// TwinCAT 3 PLC project SLAC_19046_PLC_v2
// ProgramVersion: 3.1.4023.0
// libraries:
//   Tc2_MC2, * (Beckhoff Automation GmbH)
//   Tc2_Standard, * (Beckhoff Automation GmbH)
//   Tc2_System, * (Beckhoff Automation GmbH)
//   Tc2_Utilities, * (Beckhoff Automation GmbH)
//   Tc3_Module, * (Beckhoff Automation GmbH)
// project tree:
//   / PlcTask.TcTTO
//   POUs/ AirPitch_Limit_Switches.TcPOU, AirRoll_Limit_Switches.TcPOU, AirVertical_Limit_Switches.TcPOU, CrystalGap_Limit_Switches.TcPOU, FB_Test.TcPOU, MAIN.TcPOU, YAG_LimitSwitched.TcPOU
// real-time tasks:
//   TASK PlcTask: cycle T#10ms, priority 20, ADS port 350
// motion (NC):
//   TASK NC-Task 1 SAF: cycle T#2ms, priority 4, ADS port 501
//   TASK NC-Task 1 SVB: cycle T#10ms, priority 8, ADS port 511
//   AXIS AirPitch (id 1)
//     General: UnitName=mrad
//     Dynamic: Acceleration=8.99313, Deceleration=8.99313, Jerk=27.7544
//     Velo: SlowManual=1, FastManual=2, Maximum=3.1
//     TargetPosControl: Range=0.001
//     OtherSettings: AllowMotionCmdToSlave=true, PulseDistancePos=0.5, PulseDistanceNeg=0.5
//     encoder EncType=29
//       EncPara: ScaleFactorNumerator=1.2657e-07, Offset=-4.6852, MaxCount=#xffffffff, ReferenceSystem=1
//         SoftEndMinControl: Enable=true, Range=-3.5
//         SoftEndMaxControl: Enable=true, Range=2.8
//         Inc: RefSoftSyncMask=#x0000ffff
//     drive DrvType=24
//       DrvPara: Inverse=true
//         Analog: VeloReferenz=3.3, TorqueSetpointScale=10, ScaleFactorActTorque=0.1
//         TimeComp: TaskDelayCycles=1
//     controller CtrType=3
//       CtrPara: PriorControlFactor=1
//         PosDiffControl: Range=0.5
//         PID: PosKp=10, PosTv=0.2, DeadBandPosition=0.0001
//         Observer: BandWidth=20
//   AXIS AirVert (id 2)
//     Dynamic: Acceleration=2.95205, Deceleration=2.95205, Jerk=8.98412
//     Velo: SlowManual=0.1, FastManual=0.3, Maximum=1
//     PositionAreaControl: Range=0.05
//     TargetPosControl: Range=0.0001
//     OtherSettings: AllowMotionCmdToSlave=true
//     encoder EncType=29
//       EncPara: ScaleFactorNumerator=1e-06, Offset=-10.712, MaxCount=#xffffffff
//         SoftEndMinControl: Enable=true, Range=-4.1
//         SoftEndMaxControl: Enable=true, Range=3
//         Inc: RefSoftSyncMask=#x0000ffff
//     drive DrvType=24
//       DrvPara: Inverse=true
//         Analog: VeloReferenz=3, TorqueSetpointScale=10, ScaleFactorActTorque=0.1
//         TimeComp: TaskDelayCycles=1
//     controller CtrType=3
//       CtrPara: PriorControlFactor=1
//         PosDiffControl: Range=0.15
//         PID: PosKp=7, PosTv=0.2
//         Observer: BandWidth=20
//   AXIS AirRoll (id 3)
//     General: UnitName=mrad
//     Dynamic: Acceleration=0.424188, Deceleration=0.424188, Jerk=6.42628
//     Velo: SlowManual=0.3, FastManual=1, Maximum=2.8
//     PositionAreaControl: Range=0.2
//     TargetPosControl: Range=0.0005
//     OtherSettings: AllowMotionCmdToSlave=true, PulseDistancePos=1, PulseDistanceNeg=1
//     encoder EncType=29
//       EncPara: ScaleFactorNumerator=2.4267e-07, Offset=-1031.2195, MaxCount=#xffffffff
//         SoftEndMinControl: Enable=true, Range=-4.8
//         SoftEndMaxControl: Enable=true, Range=6.1
//         Inc: RefSoftSyncMask=#x0000ffff
//     drive DrvType=24
//       Analog: VeloReferenz=3, TorqueSetpointScale=10, ScaleFactorActTorque=0.1
//       TimeComp: TaskDelayCycles=1
//     controller CtrType=3
//       CtrPara: PriorControlFactor=1
//         PosDiffControl: Range=0.5
//         PID: PosKp=10, PosTv=0.2, DeadBandPosition=0.0001
//         Observer: BandWidth=20
//   AXIS CrystalGap (id 4)
//     Dynamic: Acceleration=1.59597, Deceleration=1.59597, Jerk=4.61435
//     Velo: SlowManual=0.075, FastManual=0.2, Maximum=0.6
//     PositionAreaControl: Range=0.01
//     TargetPosControl: Range=0.0001
//     OtherSettings: AllowMotionCmdToSlave=true, PulseDistancePos=0.05, PulseDistanceNeg=0.05
//     encoder EncType=29
//       EncPara: ScaleFactorNumerator=1e-06, Offset=-19.5127, MaxCount=#xffffffff
//         SoftEndMinControl: Enable=true, Range=0.05
//         SoftEndMaxControl: Enable=true, Range=9.1
//         Inc: RefSoftSyncMask=#x0000ffff
//     drive DrvType=24
//       DrvPara: Inverse=true
//         Analog: VeloReferenz=0.3, TorqueSetpointScale=10, ScaleFactorActTorque=0.1
//         TimeComp: TaskDelayCycles=1
//     controller CtrType=3
//       CtrPara: PriorControlFactor=1
//         PosDiffControl: Range=0.15
//         PID: PosKp=4, PosTv=0.2, PosTd=1, DeadBandPosition=0.0001
//         Observer: BandWidth=20
//   AXIS YAG (id 5)
//     Dynamic: Acceleration=4.26689, Deceleration=4.26689, Jerk=19.1646
//     Velo: SlowManual=0.5, FastManual=1, Maximum=2
//     PositionAreaControl: Range=0.05
//     TargetPosControl: Range=0.05
//     OtherSettings: AllowMotionCmdToSlave=true
//     encoder EncType=29
//       EncPara: ScaleFactorNumerator=1e-06, Offset=-17, MaxCount=#xffffffff
//         SoftEndMinControl: Enable=true, Range=-0.53
//         SoftEndMaxControl: Enable=true, Range=41.6
//         Inc: RefSoftSyncMask=#x0000ffff
//     drive DrvType=24
//       Analog: VeloReferenz=20, TorqueSetpointScale=10, ScaleFactorActTorque=0.1
//       TimeComp: TaskDelayCycles=1
//     controller CtrType=3
//       CtrPara: PriorControlFactor=1
//         PosDiffControl: Range=1
//         PID: PosKp=15, PosTv=0.2, DeadBandPosition=0.01
//         Observer: BandWidth=20
//   AXIS Test (id 6)
//     TargetPosControl: Range=0.01
//     OtherSettings: AllowMotionCmdToSlave=true
//     encoder EncType=1
//     drive DrvType=5
//       Analog: TorqueSetpointScale=10, ScaleFactorActTorque=0.1
//       TimeComp: TaskDelayCycles=1
//     controller CtrType=1
//       CtrPara: PriorControlFactor=1
//         Observer: BandWidth=20
// I/O:
//   DEVICE Device 1 (EtherCAT), AmsNetId 134.79.81.23.2.1
//     Term 3 (EK1100) [EK1100 EtherCAT Coupler (2A E-Bus)]
//       Term 4 (EL7047) Air Pitch [EL7047 1Ch. Stepper motor output stage (50V, 5A)]
//       Term 5 (EL7047) Air Vertical [EL7047 1Ch. Stepper motor output stage (50V, 5A)]
//       Term 6 (EL7047) Air Roll [EL7047 1Ch. Stepper motor output stage (50V, 5A)]
//       Term 7 (EL7047) Crystal Gap [EL7047 1Ch. Stepper motor output stage (50V, 5A)]
//       Term 8 (EL7047) YAG [EL7047 1Ch. Stepper motor output stage (50V, 5A)]
//       Term 19 (EL9400) E-Bus Power Supplier [EL9400 E-Bus Power Supplier]
//       Term 9 (EL5042) Ch1 AirP Ch2 AirV [EL5042 2Ch. BiSS-C Encoder]
//       Term 10 (EL5042) Ch1 AirR Ch2 CGap [EL5042 2Ch. BiSS-C Encoder]
//       Term 11 (EL5042) Ch1 YAG [EL5042 2Ch. BiSS-C Encoder]
//       Term 13 (EL3201) Pt100 Upper Cryst [EL3201 1Ch. Ana. Input PT100 (RTD)]
//       Term 14 (EL3201) Pt100 Lower Cryst [EL3201 1Ch. Ana. Input PT100 (RTD)]
//       Term 15 (EL3201) Pt100 YAG [EL3201 1Ch. Ana. Input PT100 (RTD)]
//       Term 16 (EL3201) Pt100 Heatsink [EL3201 1Ch. Ana. Input PT100 (RTD)]
//       Term 17 (EL2634) Camera and Fan Relay [EL2634 4Ch. Relay Output, NO (250V AC / 30V DC)]
//       Term 18 (EL9011) [EL9011 End Terminal]
// variable links:
//   NC-Task 1 SAF/Axes/AirPitch <-> Device 1 (EtherCAT)/Term 3 (EK1100)/Term 4 (EL7047) Air Pitch
//     Drive/Inputs/In/nState1 @bit 3 <-> STM Status/Status/Error
//     Drive/Inputs/In/nState1 @bit 7 <-> STM Status/Status/Motor stall
//     Drive/Inputs/In/nState1 @bit 5 <-> STM Status/Status/Moving negative
//     Drive/Inputs/In/nState1 @bit 4 <-> STM Status/Status/Moving positive
//     Drive/Inputs/In/nState1 @bit 1 <-> STM Status/Status/Ready
//     Drive/Inputs/In/nState1 <-> STM Status/Status/Ready to enable
//     Drive/Inputs/In/nState1 @bit 6 <-> STM Status/Status/Torque reduced
//     Drive/Inputs/In/nState1 @bit 2 <-> STM Status/Status/Warning
//     Drive/Inputs/In/nState2 @bit 3 <-> STM Status/Status/Digital input 1
//     Drive/Inputs/In/nState2 @bit 4 <-> STM Status/Status/Digital input 2
//     Drive/Inputs/In/nState2 @bit 5 <-> STM Status/Status/Sync error
//     Drive/Inputs/In/nState2 @bit 7 <-> STM Status/Status/TxPDO Toggle
//     Drive/Inputs/In/nState4 @bit 1 <-> WcState/InputToggle
//     Drive/Inputs/In/nState4 <-> WcState/WcState
//     Drive/Outputs/Out/nCtrl1 <-> STM Control/Control/Enable
//     Drive/Outputs/Out/nCtrl1 @bit 2 <-> STM Control/Control/Reduce torque
//     Drive/Outputs/Out/nCtrl1 @bit 1 <-> STM Control/Control/Reset
//     Drive/Outputs/Out/nCtrl2 @bit 3 <-> STM Control/Control/Digital output 1
//     Drive/Outputs/Out/nDataOut2[0] <-> STM Velocity/Velocity
//   NC-Task 1 SAF/Axes/AirPitch <-> Device 1 (EtherCAT)/Term 3 (EK1100)/Term 9 (EL5042) Ch1 AirP Ch2 AirV
//     Enc/Inputs/In/nComState @bit 1 <-> WcState/InputToggle
//     Enc/Inputs/In/nComState <-> WcState/WcState
//     Enc/Inputs/In/nDataIn1 <-> FB Inputs Channel 1/Position
//     Enc/Inputs/In/nState1 @bit 12 <-> FB Inputs Channel 1/Status/Diag
//     Enc/Inputs/In/nState1 @bit 1 <-> FB Inputs Channel 1/Status/Error
//     Enc/Inputs/In/nState1 @bit 14 <-> FB Inputs Channel 1/Status/Input cycle counter
//     Enc/Inputs/In/nState1 @bit 2 <-> FB Inputs Channel 1/Status/Ready
//     Enc/Inputs/In/nState1 @bit 13 <-> FB Inputs Channel 1/Status/TxPDO State
//     Enc/Inputs/In/nState1 <-> FB Inputs Channel 1/Status/Warning
//   NC-Task 1 SAF/Axes/AirRoll <-> Device 1 (EtherCAT)/Term 3 (EK1100)/Term 10 (EL5042) Ch1 AirR Ch2 CGap
//     Enc/Inputs/In/nComState @bit 1 <-> WcState/InputToggle
//     Enc/Inputs/In/nComState <-> WcState/WcState
//     Enc/Inputs/In/nDataIn1 <-> FB Inputs Channel 1/Position
//     Enc/Inputs/In/nState1 @bit 12 <-> FB Inputs Channel 1/Status/Diag
//     Enc/Inputs/In/nState1 @bit 1 <-> FB Inputs Channel 1/Status/Error
//     Enc/Inputs/In/nState1 @bit 14 <-> FB Inputs Channel 1/Status/Input cycle counter
//     Enc/Inputs/In/nState1 @bit 2 <-> FB Inputs Channel 1/Status/Ready
//     Enc/Inputs/In/nState1 @bit 13 <-> FB Inputs Channel 1/Status/TxPDO State
//     Enc/Inputs/In/nState1 <-> FB Inputs Channel 1/Status/Warning
//   NC-Task 1 SAF/Axes/AirRoll <-> Device 1 (EtherCAT)/Term 3 (EK1100)/Term 6 (EL7047) Air Roll
//     Drive/Inputs/In/nState1 @bit 3 <-> STM Status/Status/Error
//     Drive/Inputs/In/nState1 @bit 7 <-> STM Status/Status/Motor stall
//     Drive/Inputs/In/nState1 @bit 5 <-> STM Status/Status/Moving negative
//     Drive/Inputs/In/nState1 @bit 4 <-> STM Status/Status/Moving positive
//     Drive/Inputs/In/nState1 @bit 1 <-> STM Status/Status/Ready
//     Drive/Inputs/In/nState1 <-> STM Status/Status/Ready to enable
//     Drive/Inputs/In/nState1 @bit 6 <-> STM Status/Status/Torque reduced
//     Drive/Inputs/In/nState1 @bit 2 <-> STM Status/Status/Warning
//     Drive/Inputs/In/nState2 @bit 3 <-> STM Status/Status/Digital input 1
//     Drive/Inputs/In/nState2 @bit 4 <-> STM Status/Status/Digital input 2
//     Drive/Inputs/In/nState2 @bit 5 <-> STM Status/Status/Sync error
//     Drive/Inputs/In/nState2 @bit 7 <-> STM Status/Status/TxPDO Toggle
//     Drive/Inputs/In/nState4 @bit 1 <-> WcState/InputToggle
//     Drive/Inputs/In/nState4 <-> WcState/WcState
//     Drive/Outputs/Out/nCtrl1 <-> STM Control/Control/Enable
//     Drive/Outputs/Out/nCtrl1 @bit 2 <-> STM Control/Control/Reduce torque
//     Drive/Outputs/Out/nCtrl1 @bit 1 <-> STM Control/Control/Reset
//     Drive/Outputs/Out/nCtrl2 @bit 3 <-> STM Control/Control/Digital output 1
//     Drive/Outputs/Out/nDataOut2[0] <-> STM Velocity/Velocity
//   NC-Task 1 SAF/Axes/AirVert <-> Device 1 (EtherCAT)/Term 3 (EK1100)/Term 5 (EL7047) Air Vertical
//     Drive/Inputs/In/nState1 @bit 3 <-> STM Status/Status/Error
//     Drive/Inputs/In/nState1 @bit 7 <-> STM Status/Status/Motor stall
//     Drive/Inputs/In/nState1 @bit 5 <-> STM Status/Status/Moving negative
//     Drive/Inputs/In/nState1 @bit 4 <-> STM Status/Status/Moving positive
//     Drive/Inputs/In/nState1 @bit 1 <-> STM Status/Status/Ready
//     Drive/Inputs/In/nState1 <-> STM Status/Status/Ready to enable
//     Drive/Inputs/In/nState1 @bit 6 <-> STM Status/Status/Torque reduced
//     Drive/Inputs/In/nState1 @bit 2 <-> STM Status/Status/Warning
//     Drive/Inputs/In/nState2 @bit 3 <-> STM Status/Status/Digital input 1
//     Drive/Inputs/In/nState2 @bit 4 <-> STM Status/Status/Digital input 2
//     Drive/Inputs/In/nState2 @bit 5 <-> STM Status/Status/Sync error
//     Drive/Inputs/In/nState2 @bit 7 <-> STM Status/Status/TxPDO Toggle
//     Drive/Inputs/In/nState4 @bit 1 <-> WcState/InputToggle
//     Drive/Inputs/In/nState4 <-> WcState/WcState
//     Drive/Outputs/Out/nCtrl1 <-> STM Control/Control/Enable
//     Drive/Outputs/Out/nCtrl1 @bit 2 <-> STM Control/Control/Reduce torque
//     Drive/Outputs/Out/nCtrl1 @bit 1 <-> STM Control/Control/Reset
//     Drive/Outputs/Out/nCtrl2 @bit 3 <-> STM Control/Control/Digital output 1
//     Drive/Outputs/Out/nDataOut2[0] <-> STM Velocity/Velocity
//   NC-Task 1 SAF/Axes/AirVert <-> Device 1 (EtherCAT)/Term 3 (EK1100)/Term 9 (EL5042) Ch1 AirP Ch2 AirV
//     Enc/Inputs/In/nComState @bit 1 <-> WcState/InputToggle
//     Enc/Inputs/In/nComState <-> WcState/WcState
//     Enc/Inputs/In/nDataIn1 <-> FB Inputs Channel 2/Position
//     Enc/Inputs/In/nState1 @bit 12 <-> FB Inputs Channel 2/Status/Diag
//     Enc/Inputs/In/nState1 @bit 1 <-> FB Inputs Channel 2/Status/Error
//     Enc/Inputs/In/nState1 @bit 14 <-> FB Inputs Channel 2/Status/Input cycle counter
//     Enc/Inputs/In/nState1 @bit 2 <-> FB Inputs Channel 2/Status/Ready
//     Enc/Inputs/In/nState1 @bit 13 <-> FB Inputs Channel 2/Status/TxPDO State
//     Enc/Inputs/In/nState1 <-> FB Inputs Channel 2/Status/Warning
//   NC-Task 1 SAF/Axes/CrystalGap <-> Device 1 (EtherCAT)/Term 3 (EK1100)/Term 10 (EL5042) Ch1 AirR Ch2 CGap
//     Enc/Inputs/In/nComState @bit 1 <-> WcState/InputToggle
//     Enc/Inputs/In/nComState <-> WcState/WcState
//     Enc/Inputs/In/nDataIn1 <-> FB Inputs Channel 2/Position
//     Enc/Inputs/In/nState1 @bit 12 <-> FB Inputs Channel 2/Status/Diag
//     Enc/Inputs/In/nState1 @bit 1 <-> FB Inputs Channel 2/Status/Error
//     Enc/Inputs/In/nState1 @bit 14 <-> FB Inputs Channel 2/Status/Input cycle counter
//     Enc/Inputs/In/nState1 @bit 2 <-> FB Inputs Channel 2/Status/Ready
//     Enc/Inputs/In/nState1 @bit 13 <-> FB Inputs Channel 2/Status/TxPDO State
//     Enc/Inputs/In/nState1 <-> FB Inputs Channel 2/Status/Warning
//   NC-Task 1 SAF/Axes/CrystalGap <-> Device 1 (EtherCAT)/Term 3 (EK1100)/Term 7 (EL7047) Crystal Gap
//     Drive/Inputs/In/nState1 @bit 3 <-> STM Status/Status/Error
//     Drive/Inputs/In/nState1 @bit 7 <-> STM Status/Status/Motor stall
//     Drive/Inputs/In/nState1 @bit 5 <-> STM Status/Status/Moving negative
//     Drive/Inputs/In/nState1 @bit 4 <-> STM Status/Status/Moving positive
//     Drive/Inputs/In/nState1 @bit 1 <-> STM Status/Status/Ready
//     Drive/Inputs/In/nState1 <-> STM Status/Status/Ready to enable
//     Drive/Inputs/In/nState1 @bit 6 <-> STM Status/Status/Torque reduced
//     Drive/Inputs/In/nState1 @bit 2 <-> STM Status/Status/Warning
//     Drive/Inputs/In/nState2 @bit 3 <-> STM Status/Status/Digital input 1
//     Drive/Inputs/In/nState2 @bit 4 <-> STM Status/Status/Digital input 2
//     Drive/Inputs/In/nState2 @bit 5 <-> STM Status/Status/Sync error
//     Drive/Inputs/In/nState2 @bit 7 <-> STM Status/Status/TxPDO Toggle
//     Drive/Inputs/In/nState4 @bit 1 <-> WcState/InputToggle
//     Drive/Inputs/In/nState4 <-> WcState/WcState
//     Drive/Outputs/Out/nCtrl1 <-> STM Control/Control/Enable
//     Drive/Outputs/Out/nCtrl1 @bit 2 <-> STM Control/Control/Reduce torque
//     Drive/Outputs/Out/nCtrl1 @bit 1 <-> STM Control/Control/Reset
//     Drive/Outputs/Out/nCtrl2 @bit 3 <-> STM Control/Control/Digital output 1
//     Drive/Outputs/Out/nDataOut2[0] <-> STM Velocity/Velocity
//   NC-Task 1 SAF/Axes/YAG <-> Device 1 (EtherCAT)/Term 3 (EK1100)/Term 11 (EL5042) Ch1 YAG
//     Enc/Inputs/In/nComState @bit 1 <-> WcState/InputToggle
//     Enc/Inputs/In/nComState <-> WcState/WcState
//     Enc/Inputs/In/nDataIn1 <-> FB Inputs Channel 1/Position
//     Enc/Inputs/In/nState1 @bit 12 <-> FB Inputs Channel 1/Status/Diag
//     Enc/Inputs/In/nState1 @bit 1 <-> FB Inputs Channel 1/Status/Error
//     Enc/Inputs/In/nState1 @bit 14 <-> FB Inputs Channel 1/Status/Input cycle counter
//     Enc/Inputs/In/nState1 @bit 2 <-> FB Inputs Channel 1/Status/Ready
//     Enc/Inputs/In/nState1 @bit 13 <-> FB Inputs Channel 1/Status/TxPDO State
//     Enc/Inputs/In/nState1 <-> FB Inputs Channel 1/Status/Warning
//   NC-Task 1 SAF/Axes/YAG <-> Device 1 (EtherCAT)/Term 3 (EK1100)/Term 8 (EL7047) YAG
//     Drive/Inputs/In/nState1 @bit 3 <-> STM Status/Status/Error
//     Drive/Inputs/In/nState1 @bit 7 <-> STM Status/Status/Motor stall
//     Drive/Inputs/In/nState1 @bit 5 <-> STM Status/Status/Moving negative
//     Drive/Inputs/In/nState1 @bit 4 <-> STM Status/Status/Moving positive
//     Drive/Inputs/In/nState1 @bit 1 <-> STM Status/Status/Ready
//     Drive/Inputs/In/nState1 <-> STM Status/Status/Ready to enable
//     Drive/Inputs/In/nState1 @bit 6 <-> STM Status/Status/Torque reduced
//     Drive/Inputs/In/nState1 @bit 2 <-> STM Status/Status/Warning
//     Drive/Inputs/In/nState2 @bit 3 <-> STM Status/Status/Digital input 1
//     Drive/Inputs/In/nState2 @bit 4 <-> STM Status/Status/Digital input 2
//     Drive/Inputs/In/nState2 @bit 5 <-> STM Status/Status/Sync error
//     Drive/Inputs/In/nState2 @bit 7 <-> STM Status/Status/TxPDO Toggle
//     Drive/Inputs/In/nState4 @bit 1 <-> WcState/InputToggle
//     Drive/Inputs/In/nState4 <-> WcState/WcState
//     Drive/Outputs/Out/nCtrl1 <-> STM Control/Control/Enable
//     Drive/Outputs/Out/nCtrl1 @bit 2 <-> STM Control/Control/Reduce torque
//     Drive/Outputs/Out/nCtrl1 @bit 1 <-> STM Control/Control/Reset
//     Drive/Outputs/Out/nCtrl2 @bit 3 <-> STM Control/Control/Digital output 1
//     Drive/Outputs/Out/nDataOut2[0] <-> STM Velocity/Velocity
//   SLAC_19046_PLC_v2/SLAC_19046_PLC_v2 Instance <-> Device 1 (EtherCAT)/Term 3 (EK1100)/Term 10 (EL5042) Ch1 AirR Ch2 CGap
//     PlcTask Inputs/AirRoll_Limit_Switches.fbtest.nEncoderCount <-> FB Inputs Channel 1/Position
//     PlcTask Inputs/CrystalGap_Limit_Switches.fbtest.nEncoderCount <-> FB Inputs Channel 2/Position
//   SLAC_19046_PLC_v2/SLAC_19046_PLC_v2 Instance <-> Device 1 (EtherCAT)/Term 3 (EK1100)/Term 11 (EL5042) Ch1 YAG
//     PlcTask Inputs/YAG_LimitSwitched.fbtest.nEncoderCount <-> FB Inputs Channel 1/Position
//   SLAC_19046_PLC_v2/SLAC_19046_PLC_v2 Instance <-> Device 1 (EtherCAT)/Term 3 (EK1100)/Term 4 (EL7047) Air Pitch
//     PlcTask Inputs/AirPitch_Limit_Switches.I_moter_AirPich <-> STM Synchron info data/Info data 2
//     PlcTask Inputs/AirPitch_Limit_Switches.biLimBwd_AirPitch <-> STM Status/Status/Digital input 1
//     PlcTask Inputs/AirPitch_Limit_Switches.biLimFwd_AirPitch <-> STM Status/Status/Digital input 2
//     PlcTask Inputs/AirPitch_Limit_Switches.fbtest.nMotorCurrent <-> STM Synchron info data/Info data 2
//     PlcTask Inputs/AirPitch_Limit_Switches.fbtest.nMotorLoad <-> STM Synchron info data/Info data 1
//     PlcTask Inputs/CrystalGap_Limit_Switches.biLimBwd_AirPitch <-> STM Status/Status/Digital input 1
//   SLAC_19046_PLC_v2/SLAC_19046_PLC_v2 Instance <-> Device 1 (EtherCAT)/Term 3 (EK1100)/Term 5 (EL7047) Air Vertical
//     PlcTask Inputs/AirVertical_Limit_Switches.biLimBwd_AirVertical <-> STM Status/Status/Digital input 2
//     PlcTask Inputs/AirVertical_Limit_Switches.biLimFwd_AirVertical <-> STM Status/Status/Digital input 1
//     PlcTask Inputs/AirVertical_Limit_Switches.fbtest.nMotorCurrent <-> STM Synchron info data/Info data 2
//     PlcTask Inputs/AirVertical_Limit_Switches.fbtest.nMotorLoad <-> STM Synchron info data/Info data 1
//   SLAC_19046_PLC_v2/SLAC_19046_PLC_v2 Instance <-> Device 1 (EtherCAT)/Term 3 (EK1100)/Term 6 (EL7047) Air Roll
//     PlcTask Inputs/AirRoll_Limit_Switches.biLimBwd_AirRoll <-> STM Status/Status/Digital input 1
//     PlcTask Inputs/AirRoll_Limit_Switches.biLimFwd_AirRoll <-> STM Status/Status/Digital input 2
//     PlcTask Inputs/AirRoll_Limit_Switches.fbtest.nMotorCurrent <-> STM Synchron info data/Info data 2
//     PlcTask Inputs/AirRoll_Limit_Switches.fbtest.nMotorLoad <-> STM Synchron info data/Info data 1
//     PlcTask Inputs/MAIN.biLimBwd_AirRoll <-> STM Status/Status/Digital input 2
//     PlcTask Inputs/MAIN.biLimFwd_AirRoll <-> STM Status/Status/Digital input 1
//   SLAC_19046_PLC_v2/SLAC_19046_PLC_v2 Instance <-> Device 1 (EtherCAT)/Term 3 (EK1100)/Term 7 (EL7047) Crystal Gap
//     PlcTask Inputs/CrystalGap_Limit_Switches.I_moter_Gap <-> STM Synchron info data/Info data 2
//     PlcTask Inputs/CrystalGap_Limit_Switches.biLimBwd_CrysGap <-> STM Status/Status/Digital input 1
//     PlcTask Inputs/CrystalGap_Limit_Switches.biLimFwd_CrysGap <-> STM Status/Status/Digital input 2
//     PlcTask Inputs/CrystalGap_Limit_Switches.fbtest.nMotorCurrent <-> STM Synchron info data/Info data 2
//     PlcTask Inputs/CrystalGap_Limit_Switches.fbtest.nMotorLoad <-> STM Synchron info data/Info data 1
//     PlcTask Inputs/MAIN.biLimBwd_CrysGap <-> STM Status/Status/Digital input 2
//     PlcTask Inputs/MAIN.biLimFwd_CrysGap <-> STM Status/Status/Digital input 1
//   SLAC_19046_PLC_v2/SLAC_19046_PLC_v2 Instance <-> Device 1 (EtherCAT)/Term 3 (EK1100)/Term 8 (EL7047) YAG
//     PlcTask Inputs/YAG_LimitSwitched.I_moter_Yag <-> STM Synchron info data/Info data 2
//     PlcTask Inputs/YAG_LimitSwitched.biLimBwd_YAG <-> STM Status/Status/Digital input 2
//     PlcTask Inputs/YAG_LimitSwitched.biLimFwd_YAG <-> STM Status/Status/Digital input 1
//     PlcTask Inputs/YAG_LimitSwitched.fbtest.nMotorCurrent <-> STM Synchron info data/Info data 2
//     PlcTask Inputs/YAG_LimitSwitched.fbtest.nMotorLoad <-> STM Synchron info data/Info data 1
//   SLAC_19046_PLC_v2/SLAC_19046_PLC_v2 Instance <-> Device 1 (EtherCAT)/Term 3 (EK1100)/Term 9 (EL5042) Ch1 AirP Ch2 AirV
//     PlcTask Inputs/AirPitch_Limit_Switches.fbtest.nEncoderCount <-> FB Inputs Channel 1/Position
//     PlcTask Inputs/AirVertical_Limit_Switches.fbtest.nEncoderCount <-> FB Inputs Channel 2/Position
//   SLAC_19046_PLC_v2/SLAC_19046_PLC_v2 Instance <-> NC-Task 1 SAF/Axes/AirPitch
//     PlcTask Inputs/AirPitch_Limit_Switches.axisAirPitch.NcToPlc <-> Outputs/ToPlc
//     PlcTask Outputs/AirPitch_Limit_Switches.axisAirPitch.PlcToNc <-> Inputs/FromPlc
//   SLAC_19046_PLC_v2/SLAC_19046_PLC_v2 Instance <-> NC-Task 1 SAF/Axes/AirRoll
//     PlcTask Inputs/AirRoll_Limit_Switches.axisAirRoll.NcToPlc <-> Outputs/ToPlc
//     PlcTask Outputs/AirRoll_Limit_Switches.axisAirRoll.PlcToNc <-> Inputs/FromPlc
//   SLAC_19046_PLC_v2/SLAC_19046_PLC_v2 Instance <-> NC-Task 1 SAF/Axes/AirVert
//     PlcTask Inputs/AirVertical_Limit_Switches.axisAirVertical.NcToPlc <-> Outputs/ToPlc
//     PlcTask Outputs/AirVertical_Limit_Switches.axisAirVertical.PlcToNc <-> Inputs/FromPlc
//   SLAC_19046_PLC_v2/SLAC_19046_PLC_v2 Instance <-> NC-Task 1 SAF/Axes/CrystalGap
//     PlcTask Inputs/CrystalGap_Limit_Switches.axisGAP.NcToPlc <-> Outputs/ToPlc
//     PlcTask Outputs/CrystalGap_Limit_Switches.axisGAP.PlcToNc <-> Inputs/FromPlc
//   SLAC_19046_PLC_v2/SLAC_19046_PLC_v2 Instance <-> NC-Task 1 SAF/Axes/Test
//     PlcTask Inputs/MAIN.axis.NcToPlc <-> Outputs/ToPlc
//     PlcTask Outputs/MAIN.axis.PlcToNc <-> Inputs/FromPlc
//   SLAC_19046_PLC_v2/SLAC_19046_PLC_v2 Instance <-> NC-Task 1 SAF/Axes/YAG
//     PlcTask Inputs/YAG_LimitSwitched.axisYAG.NcToPlc <-> Outputs/ToPlc
//     PlcTask Outputs/YAG_LimitSwitched.axisYAG.PlcToNc <-> Inputs/FromPlc

CONFIGURATION SLAC_19046_PLC_v2
    RESOURCE PLC ON TwinCAT3
        TASK PlcTask(INTERVAL := T#10ms, PRIORITY := 20);
        PROGRAM MAIN WITH PlcTask : MAIN;
    END_RESOURCE
END_CONFIGURATION

// ---- POUs/MAIN.TcPOU
PROGRAM MAIN
VAR
    axis: AXIS_REF;
    fbAxisPower: MC_Power;
    //fbAxisMoveAbsolute: MC_MoveAbsolute;
    
	bEnable: BOOL := TRUE;
	Enable_Positive: BOOL:= TRUE;
	Enable_Negative: BOOL:= TRUE;
    fOverride: LREAL := 100;
    	
	biLimFwd_AirRoll AT %I*: BOOL;
	biLimBwd_AirRoll AT %I*: BOOL;
	
	biLimFwd_CrysGap AT %I*: BOOL;
	biLimBwd_CrysGap AT %I*: BOOL;
	
	fbtestMain:FB_TEST;
	fbtestSelection:FB_TEST;
	iTestStageID:int:=0;
	
	
	fbScopeServerControl: FB_ScopeServerControl;
   eReqState: E_ScopeServerState := SCOPE_SERVER_IDLE;
	
END_VAR

(*This is only used for the scope purposes, so we don't have to change the aquisition axis everytime 
we switch test between access*)

CASE iTestStageID OF
	0: //test axis
		fbtestSelection := fbtestMain;
	1: //Air Pitch
		fbtestSelection := AirPitch_Limit_Switches.fbtest;
	2://Air Roll
		fbtestSelection := AirRoll_Limit_Switches.fbtest;
	3: //Air Vertical
    	fbtestSelection := AirVertical_Limit_Switches.fbtest;
	4: // In Vac YAG
		fbtestSelection := YAG_LimitSwitched.fbtest;
	5: // In Vac Gap
		fbtestSelection := CrystalGap_Limit_Switches.fbtest;
END_CASE

AirPitch_Limit_Switches();
AirRoll_Limit_Switches();
AirVertical_Limit_Switches();
YAG_LimitSwitched();
CrystalGap_Limit_Switches();


fbtestMain(
	axis:=axis , 
	fTargetVelocity:=1 , 
	fStartPosition:= 0.5, 
	fEndPosition:= 10, 
	nDivisions:= 5 , 
	bRunAll:=TRUE,
	fbAxisPower:= fbAxisPower );

Enable_Positive:= (axis.NcToPlc.ActPos <10);
Enable_Negative := (axis.NcToPlc.ActPos >0.5);

fbAxisPower(
    Axis:= axis,
    Enable:= bEnable,
    Enable_Positive:= Enable_Positive,
    Enable_Negative:= Enable_Negative,
    Override:= fOverride,
    BufferMode:= ,
    Options:= ,
    Status=> ,
    Busy=> ,
    Active=> ,
    Error=> ,
    ErrorID=> );

END_PROGRAM

// ---- POUs/FB_Test.TcPOU
FUNCTION_BLOCK FB_Test


VAR_INPUT
	fTargetVelocity: LREAL := 0.1;
	fPositionDelta:LREAL := 0.009;
	fStartPosition: LREAL := 0; //Negative
	fEndPosition: LREAL := 0; //Positive
	nDivisions: int := 1;
	bRunAll:BOOL:=FALSE;
END_VAR



VAR_IN_OUT
	axis: AXIS_REF;
	fbAxisPower: MC_Power;
	
END_VAR

VAR
	
	fbAxisMoveAbsolute: MC_MoveAbsolute;
	
	
	bMove: BOOL := FALSE;
	fTargetPosition: LREAL := 0;
	rActPosLimBwd_AirPitch: LREAL;
	rSetPosLimBwd_AirPitch: LREAL;
	step: INT;


	fOverride: LREAL := 100;
	bEnable: BOOL := FALSE;
	nStep: int := 0; // set to 1 to start the step test, 7 full stroke, 20 HL rep test, 30 LL rep test
	nCount: int := 0;
	fPositionInc: LREAL;
	
	tWait: TON;
	tTimeout: TON; //timeout
	bError:BOOL :=FALSE;
	bTestComplete:BOOL:=FALSE;
	rMinPosDiff: LREAL :=1000;
	fMaxPosDiff: LREAL:=-1000;
	
	rActPosLimFwd:LREAL; //save the actual motor position
	rActPosLimBwd:LREAL;
	
	rEncPosLimFwd:LREAL; //save the actual motor position
	rEncPosLimBwd:LREAL;
	
	rSetPosLimFwd:LREAL; //save the set motor position
	rSetPosLimBwd:LREAL;
	
	aPosLimFwd: ARRAY[1..5] OF LREAL;
	aPosLimBwd: ARRAY[1..5] OF LREAL;
	aEncLimFwd: ARRAY[1..5] OF LREAL;
	aEncLimBwd: ARRAY[1..5] OF LREAL;
	index:int:=0;
	
	ftLimFwd :F_TRIG; //detect falling edge on the limit switch
	ftLimBwd :F_TRIG;
	
	nMotorLoad AT %I*: UINT; //default Info data 1
	nMotorCurrent AT %I*: UINT;//default info data 2
	nEncoderCount AT %I*: ULINT;
	
	fbScopeServerControl: FB_ScopeServerControl;
   eReqState: E_ScopeServerState := SCOPE_SERVER_IDLE;
END_VAR

axis.ReadStatus();




fbAxisMoveAbsolute(
	Axis:= axis,
	Execute:= bMove,
	Position:= fTargetPosition,
	Velocity:= fTargetVelocity,
	Acceleration:= ,
	Deceleration:= ,
	Jerk:= ,
	BufferMode:= ,
	Options:= ,
	Done=> ,
	Busy=> ,
	Active=> ,
	CommandAborted=> ,
	Error=> ,
	ErrorID=> );
	
	
	CASE nStep OF
		
		0: 
			bEnable:=FALSE;
			bMove:=FALSE;
			nCount:=0;
			IF (nDivisions <> 0) THEN
				fPositionInc := (fEndPosition -fStartPosition) /nDivisions;
			END_IF
			//eReqState:= E_ScopeServerState.SCOPE_SERVER_STOP;
			 

		1:
			eReqState:= E_ScopeServerState.SCOPE_SERVER_CONNECT;
			eReqState:= E_ScopeServerState.SCOPE_SERVER_START;
			bTestComplete := FALSE;
			bError:=FALSE;
			bEnable:= TRUE;
			IF (fbAxisPower.Status) THEN
				nStep:=nStep+1;
			END_IF;
			
			
		2:
			fTargetPosition := fStartPosition;
			bMove:= TRUE;
			nStep:=nStep+1;
			IF fbAxisMoveAbsolute.Active THEN
				bMove:=FALSE;
				nStep:=nStep+1;
			END_IF
			
		3:
			IF (*fbAxisMoveAbsolute.Done AND*) tWait.Q (*(axis.Status.InTargetPosition)*) THEN
				fTargetPosition := fbAxisMoveAbsolute.Position + fPositionInc;
				nStep:=nStep+1;
				bMove:=FALSE;
				IF ( fTargetPosition > fEndPosition )  THEN 
				fTargetPosition:= fEndPosition;
				END_IF
			END_IF
			IF (axis.NcToPlc.ActPos >= fEndPosition-fPositionDelta) THEN 
					nStep:=5;
			END_IF
			//IF (fbAxisMoveAbsolute.Error) THEN
			//	nStep:=999;
			//END_IF
		
		4:
			bMove:= TRUE;
			IF fbAxisMoveAbsolute.Active THEN
				bMove:=FALSE;
				nStep:=3;	
			
			END_IF
		
			
		5:
			IF (*fbAxisMoveAbsolute.Done AND*) tWait.Q (* (axis.Status.InTargetPosition)*) THEN
				fTargetPosition := fbAxisMoveAbsolute.Position - fPositionInc;
				nStep:=nStep+1;
				bMove:=FALSE;
				IF ( fTargetPosition < fStartPosition )  THEN 
				fTargetPosition:= fStartPosition;
				END_IF
			END_IF
			IF (axis.NcToPlc.ActPos <= fStartPosition+fPositionDelta) THEN
				IF NOT(bRunAll) THEN nStep:=0; ELSE nStep:=7; END_IF
				bTestComplete := TRUE;
			END_IF
		
		6:
			bMove:= TRUE;
			IF fbAxisMoveAbsolute.Active THEN
				bMove:=FALSE;
				nStep:=5;	
			END_IF
			
		7: // Full stroke, the stage is back to the start position, move to the end position
			bTestComplete := FALSE;
			bError:=FALSE;
			fTargetPosition := fEndPosition;
			bMove:= TRUE;
			IF fbAxisMoveAbsolute.Active OR (axis.NcToPlc.ActPos >= fEndPosition-fPositionDelta)THEN
				bMove:=FALSE;
				nStep:=nStep+1;
			END_IF
		8: // wait until the stage is at the end position then set position to start position
		  IF (*fbAxisMoveAbsolute.Done AND*) tWait.Q (*(axis.Status.InTargetPosition)*) OR (axis.NcToPlc.ActPos >= fEndPosition-fPositionDelta) THEN
				fTargetPosition := fStartPosition;
				nStep:=nStep+1;
				bMove:=FALSE;
			END_IF
		9: //Activate move
			bMove:= TRUE;
			IF fbAxisMoveAbsolute.Active THEN
				bMove:=FALSE;
				nStep:=nStep+1;	
			END_IF
		 10:// wait until the stage reaches the start position
		   IF (*fbAxisMoveAbsolute.Done AND*) tWait.Q (*(axis.Status.InTargetPosition)*) THEN
				fTargetPosition := fStartPosition;
				IF NOT(bRunAll) THEN nStep:=0; ELSE nStep:=20; END_IF
				bTestComplete := TRUE;
				bMove:=FALSE;
			END_IF

		20:  //High Limit switch repitition test
			index:=1;
			nStep:=nStep+1;
			
		21: //High Limit switch repitition test
			bTestComplete := FALSE;
			bError:=FALSE;
			fTargetPosition := fEndPosition;
			bMove:= TRUE;
			IF fbAxisMoveAbsolute.Active OR (axis.NcToPlc.ActPos >= fEndPosition-fPositionDelta)THEN
				bMove:=FALSE;
				nStep:=nStep+1;
			END_IF
		22: // wait until the stage is at the end position
		  IF (*fbAxisMoveAbsolute.Done AND*) tWait.Q (*(axis.Status.InTargetPosition)*) OR fbAxisPower.Enable_Positive  THEN
				fTargetPosition := fEndPosition - fPositionInc;
				aPosLimFwd[index]:= rActPosLimFwd;
				aEncLimFwd[index]:= rEncPosLimFwd;
				index:=index+1;
				nStep:=nStep+1;
				bMove:=FALSE;
			END_IF
		23: //Activate move
			bMove:= TRUE;
			IF fbAxisMoveAbsolute.Active THEN
				bMove:=FALSE;
				nStep:=nStep+1;	
			END_IF
		24: // wait until the stage is at the end position
		  IF (*fbAxisMoveAbsolute.Done AND*) tWait.Q (*(axis.Status.InTargetPosition)*) THEN
				fTargetPosition := fEndPosition;
				if (index<=5) THEN nStep:=21; ELSE IF NOT(bRunAll) THEN nStep:=0; ELSE nStep:=30; END_IF END_IF
				bMove:=FALSE;
			END_IF
		
			
			
		30: // Low Limit Switch rep
			index:=1;
			nStep:=nStep+1;
			
		31: //Low Limit switch repitition test
			bTestComplete := FALSE;
			bError:=FALSE;
			fTargetPosition := fStartPosition;
			bMove:= TRUE;
			
			IF fbAxisMoveAbsolute.Active OR (axis.NcToPlc.ActPos <= fStartPosition+fPositionDelta)THEN
				bMove:=FALSE;
				nStep:=nStep+1;
			END_IF
		32: // wait until the stage is at the end position
		  IF (*fbAxisMoveAbsolute.Done AND*) tWait.Q (*(axis.Status.InTargetPosition)*) OR fbAxisPower.Enable_Negative  THEN
				fTargetPosition := fStartPosition + fPositionInc;
				aPosLimBwd[index]:= rActPosLimBwd;
				aEncLimBwd[index]:= rEncPosLimBwd;
				index:=index+1;
				nStep:=nStep+1;
				bMove:=FALSE;
			END_IF
		33: //Activate move
			bMove:= TRUE;
			IF fbAxisMoveAbsolute.Active THEN
				bMove:=FALSE;
				nStep:=nStep+1;	
			END_IF
		34: // wait until the stage is at the end position
		  IF (*fbAxisMoveAbsolute.Done AND*) tWait.Q (*(axis.Status.InTargetPosition)*) THEN
				fTargetPosition := fEndPosition;
				if (index<=5) THEN nStep:=31; ELSE nStep:=0; END_IF
				bMove:=FALSE;
			END_IF
		
	
	END_CASE
	
tWait(In:= axis.Status.InTargetPosition, PT:=T#2S);
tTimeout(In:= (step = 3) OR (step =5), PT:=T#5S);


IF (tTimeout.Q ) OR (fbAxisMoveAbsolute.Error) THEN bError:=TRUE; step:=0; END_IF;	
axis.ReadStatus();
//fbAxisPower(Enable := bEnable);



// Saving limit switches positions
ftLimFwd(CLK:= fbAxisPower.Enable_Positive);
ftLimBwd(CLK:= fbAxisPower.Enable_Negative);

IF (ftLimFwd.Q) THEN
	rActPosLimFwd := axis.NcToPlc.ActPos ;
	rSetPosLimFwd := axis.NcToPlc.SetPos;
	rEncPosLimFwd := axis.NcToPlc.ActPos ;
END_IF

IF (ftLimBwd.Q) THEN
	rActPosLimBwd := axis.NcToPlc.ActPos ;
	rSetPosLimBwd:= axis.NcToPlc.SetPos;
	rEncPosLimBwd := axis.NcToPlc.ActPos ;
END_IF


// Saving Min and Max position diff
IF (axis.NcToPlc.PosDiff < rMinPosDiff) THEN rMinPosDiff := axis.NcToPlc.PosDiff; END_IF
IF (axis.NcToPlc.PosDiff > fMaxPosDiff) THEN fMaxPosDiff := axis.NcToPlc.PosDiff; END_IF
(*
fbScopeServerControl(
   sNetId:= '127.0.0.1.1.1',
   eReqState:= eReqState,
   sConfigFile:= 'C:\GitHub\Exit-Slits\Measurement Project\Scope Project1.tcscopex',
   sSaveFile:= 'C:\GitHub\Exit-Slits\FAT Scopes\test.svd',
   tTimeout:= t#5s,
   bBusy=>,
   bDone=>,
   bError=>,
   nErrorId=>);*)

END_FUNCTION_BLOCK

// ---- POUs/AirPitch_Limit_Switches.TcPOU
PROGRAM AirPitch_Limit_Switches

VAR
	
 	axisAirPitch: AXIS_REF;
    fbAxisPowerAirPitch: MC_Power;
       
	bEnable: BOOL := TRUE;
    fOverride: LREAL := 100;
    		
	biLimFwd_AirPitch AT %I*: BOOL;
	biLimBwd_AirPitch AT %I*: BOOL;

	fbtest:FB_Test;
	I_moter_AirPich AT %I*: UINT;

END_VAR



fbtest(
	axis:=axisAirPitch , 
	fTargetVelocity:=0.12 , 
	fStartPosition:= -3.7 , 
	fEndPosition:= 3, 
	nDivisions:= 20 , 
	fbAxisPower:= fbAxisPowerAirPitch );

fbAxisPowerAirPitch(
    Axis:= axisAirPitch,
    Enable:= bEnable,
    Enable_Positive:= biLimFwd_AirPitch, // TRUE, //
    Enable_Negative:= biLimBwd_AirPitch, // TRUE, //
    Override:= fOverride,
    BufferMode:= ,
    Options:= ,
    Status=> ,
    Busy=> ,
    Active=> ,
    Error=> ,
    ErrorID=> );

END_PROGRAM

// ---- POUs/AirRoll_Limit_Switches.TcPOU
PROGRAM AirRoll_Limit_Switches

VAR
 	axisAirRoll: AXIS_REF;
    fbAxisPowerAirRoll: MC_Power;
       
	bEnable: BOOL := TRUE;
    fOverride: LREAL := 100;
    		
	biLimFwd_AirRoll AT %I*: BOOL;
	biLimBwd_AirRoll AT %I*: BOOL;
	
	fbtest:FB_Test;

END_VAR


fbtest(
	axis:=axisAirRoll , 
	fTargetVelocity:=0.24 , 
	fStartPosition:= -4.82, 
	fEndPosition:= 6.22 , 
	nDivisions:= 20 , 
	fbAxisPower:= fbAxisPowerAirRoll );

fbAxisPowerAirRoll(
    Axis:= axisAirRoll,
    Enable:= bEnable,
    Enable_Positive:= biLimFwd_AirRoll, // TRUE, //
    Enable_Negative:= biLimBwd_AirRoll, // TRUE, //
    Override:= fOverride,
    BufferMode:= ,
    Options:= ,
    Status=> ,
    Busy=> ,
    Active=> ,
    Error=> ,
    ErrorID=> );

END_PROGRAM

// ---- POUs/AirVertical_Limit_Switches.TcPOU
PROGRAM AirVertical_Limit_Switches

VAR
	
	axisAirVertical: AXIS_REF;
    fbAxisPowerAirVertical: MC_Power;
       
	bEnable: BOOL := TRUE;
    fOverride: LREAL := 100;
    		
	biLimFwd_AirVertical AT %I*: BOOL;
	biLimBwd_AirVertical AT %I*: BOOL;

	fbtest:FB_Test;
END_VAR


fbtest(
	axis:=axisAirVertical , 
	fTargetVelocity:=0.3 , 
	fStartPosition:= -4.13,//-4.1, 
	fEndPosition:= 3,//3, 
	nDivisions:= 20 , 
	fbAxisPower:= fbAxisPowerAirVertical );
fbAxisPowerAirVertical(
    Axis:= axisAirVertical,
    Enable:= bEnable,
    Enable_Positive:= biLimFwd_AirVertical, // TRUE, //
    Enable_Negative:= biLimBwd_AirVertical, // TRUE, //
    Override:= fOverride,
    BufferMode:= ,
    Options:= ,
    Status=> ,
    Busy=> ,
    Active=> ,
    Error=> ,
    ErrorID=> );

END_PROGRAM

// ---- POUs/YAG_LimitSwitched.TcPOU
PROGRAM YAG_LimitSwitched

VAR
	
    axisYAG: AXIS_REF;
    fbAxisPowerYAG: MC_Power;
       
	bEnable: BOOL := TRUE;
    fOverride: LREAL := 100;
    		
	biLimFwd_YAG AT %I*: BOOL;
	biLimBwd_YAG AT %I*: BOOL;

	fbtest: FB_TEST;
	I_moter_Yag AT %I*: UINT;
	
END_VAR

fbtest(
	axis:=axisYAG , 
	fTargetVelocity:=0.2 , //0.5
	fStartPosition:= -0.53,//0, 
	fEndPosition:= 41.4,//41, 
	nDivisions:= 20 , 
	fPositionDelta:= 0.0099,
	fbAxisPower:= fbAxisPowerYAG );
fbAxisPowerYAG(
    Axis:= axisYAG,
    Enable:= bEnable,
    Enable_Positive:= biLimFwd_YAG, // TRUE, //
    Enable_Negative:= biLimBwd_YAG, // TRUE, //
    Override:= fOverride,
    BufferMode:= ,
    Options:= ,
    Status=> ,
    Busy=> ,
    Active=> ,
    Error=> ,
    ErrorID=> );

END_PROGRAM

// ---- POUs/CrystalGap_Limit_Switches.TcPOU
PROGRAM CrystalGap_Limit_Switches

VAR
	
    axisGAP: AXIS_REF;
    fbAxisPowerGAP: MC_Power;
       
	bEnable: BOOL := TRUE;
    fOverride: LREAL := 100;
    		
	biLimFwd_CrysGap AT %I*: BOOL;
	biLimBwd_CrysGap AT %I*: BOOL;
	
	fbtestGAP:FB_TEST;
	
	ftLimFwd :F_TRIG; //detect falling edge on the limit switch
	
	ftLimBwd :F_TRIG;
	
	rActPosLimFwd:LREAL; //save the actual motor position
	rActPosLimBwd:LREAL;
	
	rSetPosLimFwd:LREAL; //save the set motor position
	rSetPosLimBwd:LREAL;

// Stuff for testing cage deflection 			

	biLimFwd_AirPitch AT %I*: BOOL;
	biLimBwd_AirPitch AT %I*: BOOL;
	
	ftLimFwd_AirPitch :F_TRIG; //detect falling edge on the limit switch
	ftLimBwd_AirPitch :F_TRIG;
	
	rActPosLimFwd_AirPitch:LREAL; //save the actual motor position
	rActPosLimBwd_AirPitch:LREAL;
	
	rSetPosLimFwd_AirPitch:LREAL; //save the set motor position
	rSetPosLimBwd_AirPitch:LREAL;
		
	fbtest: FB_TEST;
	
	I_moter_Gap AT %I*: UINT;
	
END_VAR


fbtest(
	axis:=axisGAP , 
	fTargetVelocity:=0.1 , 
	fStartPosition:= 1,//0.05, 
	fEndPosition:= 4, 
	nDivisions:= 20 , 
	fbAxisPower:= fbAxisPowerGAP );


fbAxisPowerGAP(
    Axis:= axisGAP,
    Enable:= bEnable,
    Enable_Positive:= biLimFwd_CrysGap, //biLimFwd_CrysGap, //  // biLimFwd_CrysGap, // TRUE, //
    Enable_Negative:= biLimBwd_CrysGap, // TRUE, //
    Override:= fOverride,
    BufferMode:= ,
    Options:= ,
    Status=> ,
    Busy=> ,
    Active=> ,
    Error=> ,
    ErrorID=> );
	
	
//fbtestGAP(axis := axisGAP, fbAxisPower:=fbAxisPowerGAP);

ftLimFWd(CLK:= biLimFwd_CrysGap);
ftLimBwd(CLK:= biLimBwd_CrysGap);


IF (ftLimFwd.Q) THEN
	rActPosLimFwd := axisGAP.NcToPlc.ActPos ;
	rSetPosLimFwd := axisGap.NcToPlc.SetPos;
END_IF

IF (ftLimBwd.Q) THEN
	rActPosLimBwd := axisGAP.NcToPlc.ActPos ;
	rSetPosLimBwd := axisGap.NcToPlc.SetPos;
END_IF



// Stuff for testing cage deflection 	

ftLimFwd_AirPitch(CLK:= biLimFwd_AirPitch);
ftLimBwd_AirPitch(CLK:= biLimBwd_AirPitch);

IF (ftLimFwd_AirPitch.Q) THEN
	rActPosLimFwd_AirPitch := axisGAP.NcToPlc.ActPos ;
	rSetPosLimFwd_AirPitch := axisGap.NcToPlc.SetPos;
END_IF

IF (ftLimBwd_AirPitch.Q) THEN
	rActPosLimBwd_AirPitch := axisGAP.NcToPlc.ActPos ;
	rSetPosLimBwd_AirPitch := axisGap.NcToPlc.SetPos;
END_IF

END_PROGRAM
